// TIA Portal V15.1 export
// export: Created 2026-01-15T16:29:45.5741419Z, ExportSetting WithDefaults, WithReadOnly, DisplayName Totally Integrated Automation Portal, DisplayVersion V15.1 Update 8, DisplayName TIA Portal Openness, DisplayVersion V15.1 Update 8, DisplayName STEP 7 Professional, DisplayVersion V15.1 Update 8, DisplayName WinCC Advanced, DisplayVersion V15.1 Update 8
DATA_BLOCK "10.3.SKSL_1"   // DB1009
{ S7_Optimized_Access := 'TRUE' }
VERSION : 0.1
// stored: AutoNumber false, CodeModifiedDate 2026-01-15T16:25:55.7623037Z, CompileDate 2026-01-15T16:25:55.7683704Z, CreationDate 2026-01-15T16:22:49.8270549Z, DBAccessibleFromOPCUA true, DownloadWithoutReinit false, InstanceOfName 10.TIMER_CLOCK, InstanceOfNumber 10, InstanceOfType FB, InterfaceModifiedDate 2023-08-14T08:08:19.3737097Z, IsConsistent true, IsKnowHowProtected false, IsRetainMemResEnabled false, MemoryReserve 100, ModifiedDate 2026-01-15T16:25:55.7623037Z, ParameterModified 2022-05-24T16:04:05.0982286Z, StructureModified 2023-08-14T08:08:19.3737097Z, UDAEnableTagReadback false
"10.TIMER_CLOCK"
   // VAR_INPUT
   //    ON : Bool;
   //    CLOCK_1S : Bool;
   //    T_ON : Real;
   //    T_OFF : Real;
   // END_VAR
   // VAR_OUTPUT
   //    OUT : Bool;
   // END_VAR
   // VAR RETAIN
   //    TON : Real;
   //    TOFF : Real;
   // END_VAR
   // VAR
   //    CLK1 : Bool;
   // END_VAR
BEGIN
END_DATA_BLOCK
